// TIA Portal project "Controle esteira transportadora" (V14)

(* hardware
DEVICE "S71500/ET200MP station_1"  S7-1500 station
   slot 0: "Rail_0"  Rack  6ES7 590-1***0-0AA0
   slot 1: "PLC_1"  CPU 1511C-1 PN  6ES7 511-1CK00-0AB0  V2.1
      slot 3: "CPU display_1"  6ES7591-1AA00-0AA0
*)

// ===== PLC "PLC_1"  CPU 1511C-1 PN =====

DATA_BLOCK "Entradas"   // DB1
{ S7_Optimized_Access := 'TRUE' }
VERSION : 0.1
   VAR
      S1 : Bool;   // Sensor de presença
      S2 : Int;   // Sensor de tamanho
      Start : Bool;   // Inicia o sistema
      EmergenciaStop : Bool;   // Parar o sistema
      ResetContagem : Bool;   // operador pegou o lote
   END_VAR
BEGIN
END_DATA_BLOCK

DATA_BLOCK "Saidas"   // DB2
{ S7_Optimized_Access := 'TRUE' }
VERSION : 0.1
   VAR
      Motor : Bool;   // Liga Esteira
      Desviador : Bool;   // Desvia peças grandes
      Alarme : Bool;   // Alarme de se atingir 5 peças grandes
   END_VAR
BEGIN
END_DATA_BLOCK

// folder: System blocks/Program resources

DATA_BLOCK "IEC_Timer_0_DB"   // DB3
{ S7_Optimized_Access := 'TRUE' }
AUTHOR : Simatic
FAMILY : IEC
NAME : IEC_TMR
VERSION : 1.0
// stored: InstanceOfName IEC_TIMER
"IEC_TIMER"
BEGIN
END_DATA_BLOCK

DATA_BLOCK "IEC_Counter_0_DB"   // DB4
{ S7_Optimized_Access := 'TRUE' }
AUTHOR : Simatic
FAMILY : IEC
NAME : CNTR
VERSION : 1.0
// stored: InstanceOfName IEC_COUNTER
"IEC_COUNTER"
BEGIN
END_DATA_BLOCK

// folder: (top level)

FUNCTION "Controle Produto" : Void   // FC1, LAD
{ S7_Optimized_Access := 'TRUE' }
VERSION : 0.1
   VAR_INPUT
      Start : Bool;
      Stop : Bool;
      ResetContagem : Bool;
      "Sensor de Presença" : Bool;
      "Sensor de Altura" : Int;
   END_VAR
   VAR_OUTPUT
      Esteira : Bool;
      Desviador : Bool;
      Alarme : Bool;
   END_VAR
   VAR_TEMP
      EmProcesso : Bool;
      memBordaP : Bool;
      produto : Int;
   END_VAR
   VAR_TEMP   // added for the SCL form of the ladder/FBD networks
      _w1 : Bool;
      _w2 : Bool;
   END_VAR
BEGIN

REGION Network 1: Controle de processo inicialização
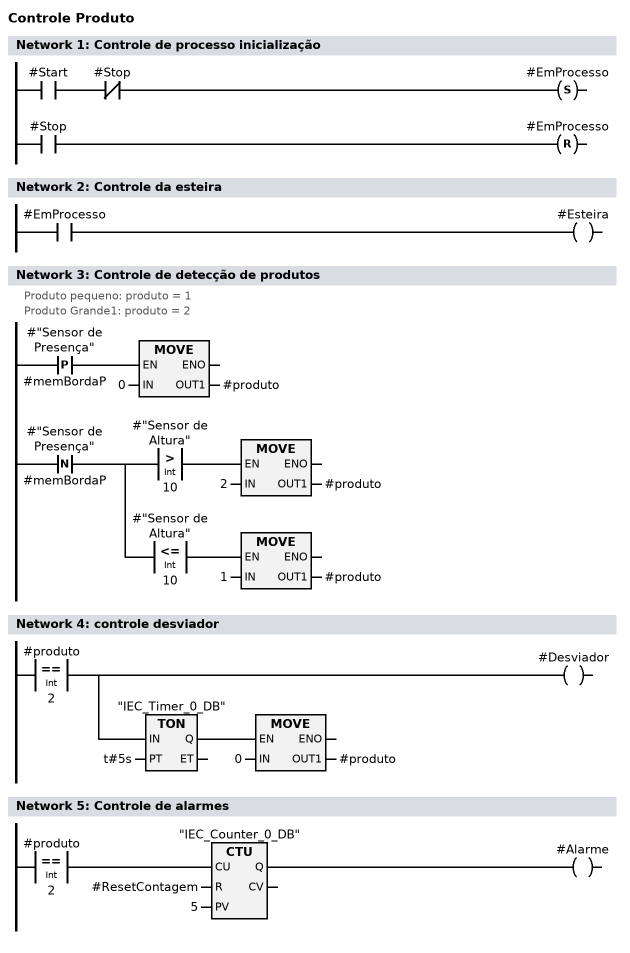
   RUNG wire#powerrail
      Contact( #Start )
      I_Contact( #Stop )
      S_Coil( #EmProcesso )
   END_RUNG
   RUNG wire#powerrail
      Contact( #Stop )
      R_Coil( #EmProcesso )
   END_RUNG
   // the same network as SCL:
   IF #Start AND NOT #Stop THEN #EmProcesso := TRUE; END_IF;
   IF #Stop THEN #EmProcesso := FALSE; END_IF;
END_REGION

REGION Network 2: Controle da esteira
   RUNG wire#powerrail
      Contact( #EmProcesso )
      Coil( #Esteira )
   END_RUNG
   // the same network as SCL:
   #Esteira := #EmProcesso;
END_REGION

REGION Network 3: Controle de detecção de produtos
   // Produto pequeno: produto = 1
   // Produto Grande1: produto = 2
   RUNG wire#powerrail
      P_Contact(operand := #"Sensor de Presença", bit := #memBordaP)
      Move(in := 0, out1 => #produto)
   END_RUNG
   RUNG wire#powerrail
      N_Contact(operand := #"Sensor de Presença", bit := #memBordaP)
      wire#w1
      { S7_Templates := "SrcType := Int" } GT_Contact(in1 := #"Sensor de Altura", in2 := 10)
      Move(in := 2, out1 => #produto)
   END_RUNG
   RUNG wire#w1
      { S7_Templates := "SrcType := Int" } LE_Contact(in1 := #"Sensor de Altura", in2 := 10)
      Move(in := 1, out1 => #produto)
   END_RUNG
   // the same network as SCL:
   #_w1 := #"Sensor de Presença" AND NOT #memBordaP;   // rising edge of #"Sensor de Presença"
   #memBordaP := #"Sensor de Presença";
   IF #_w1 THEN #produto := 0; END_IF;
   #_w2 := NOT #"Sensor de Presença" AND #memBordaP;   // falling edge of #"Sensor de Presença"
   #memBordaP := #"Sensor de Presença";
   IF #_w2 AND (#"Sensor de Altura" > 10) THEN #produto := 2; END_IF;
   IF #_w2 AND (#"Sensor de Altura" <= 10) THEN #produto := 1; END_IF;
END_REGION

REGION Network 4: controle desviador
   #Desviador := #produto = 2;
   "IEC_Timer_0_DB".TON(IN := #Desviador, PT := t#5s);
   IF "IEC_Timer_0_DB".Q THEN #produto := 0; END_IF;
END_REGION

REGION Network 5: Controle de alarmes
   "IEC_Counter_0_DB".CTU(CU := #produto = 2, R := #ResetContagem, PV := 5);
   #Alarme := "IEC_Counter_0_DB".Q;
END_REGION
END_FUNCTION

ORGANIZATION_BLOCK "Main"   // OB1, LAD, ProgramCycle
TITLE = "Main Program Sweep (Cycle)"
{ S7_Optimized_Access := 'TRUE' }
VERSION : 0.1
   VAR_INPUT
      Initial_Call : Bool;   // Initial call of this OB
      Remanence : Bool;   // =True, if remanent data are available
   END_VAR
BEGIN

REGION Network 1
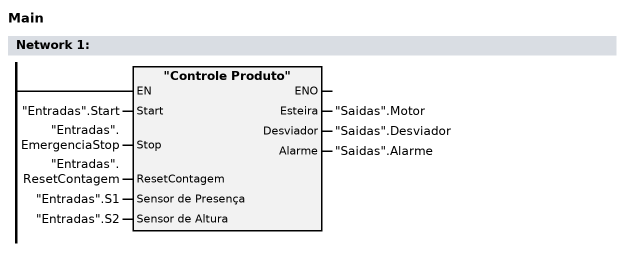
   RUNG wire#powerrail
      "Controle Produto"(Start := "Entradas".Start, Stop := "Entradas".EmergenciaStop, ResetContagem := "Entradas".ResetContagem, "Sensor de Presença" := "Entradas".S1, "Sensor de Altura" := "Entradas".S2, Esteira => "Saidas".Motor, Desviador => "Saidas".Desviador, Alarme => "Saidas".Alarme)
   END_RUNG
   // the same network as SCL:
   "Controle Produto"(Start := "Entradas".Start,
                      Stop := "Entradas".EmergenciaStop,
                      ResetContagem := "Entradas".ResetContagem,
                      "Sensor de Presença" := "Entradas".S1,
                      "Sensor de Altura" := "Entradas".S2,
                      Esteira => "Saidas".Motor,
                      Desviador => "Saidas".Desviador,
                      Alarme => "Saidas".Alarme);
END_REGION
END_ORGANIZATION_BLOCK